// TIA Portal V20 export
FUNCTION "01 T4 LANT Alarms" : Void   // FC1112, LAD
TITLE = ALARMS
{ S7_Optimized_Access := 'TRUE' }
// stored: AutoNumber false, IsIECCheckEnabled true, SetENOAutomatically false
   VAR_TEMP
      Trash : Bool;
   END_VAR
BEGIN

REGION Network 1: ============ ALARMS RESET ============
END_REGION

REGION Network 2: Alarms Reset
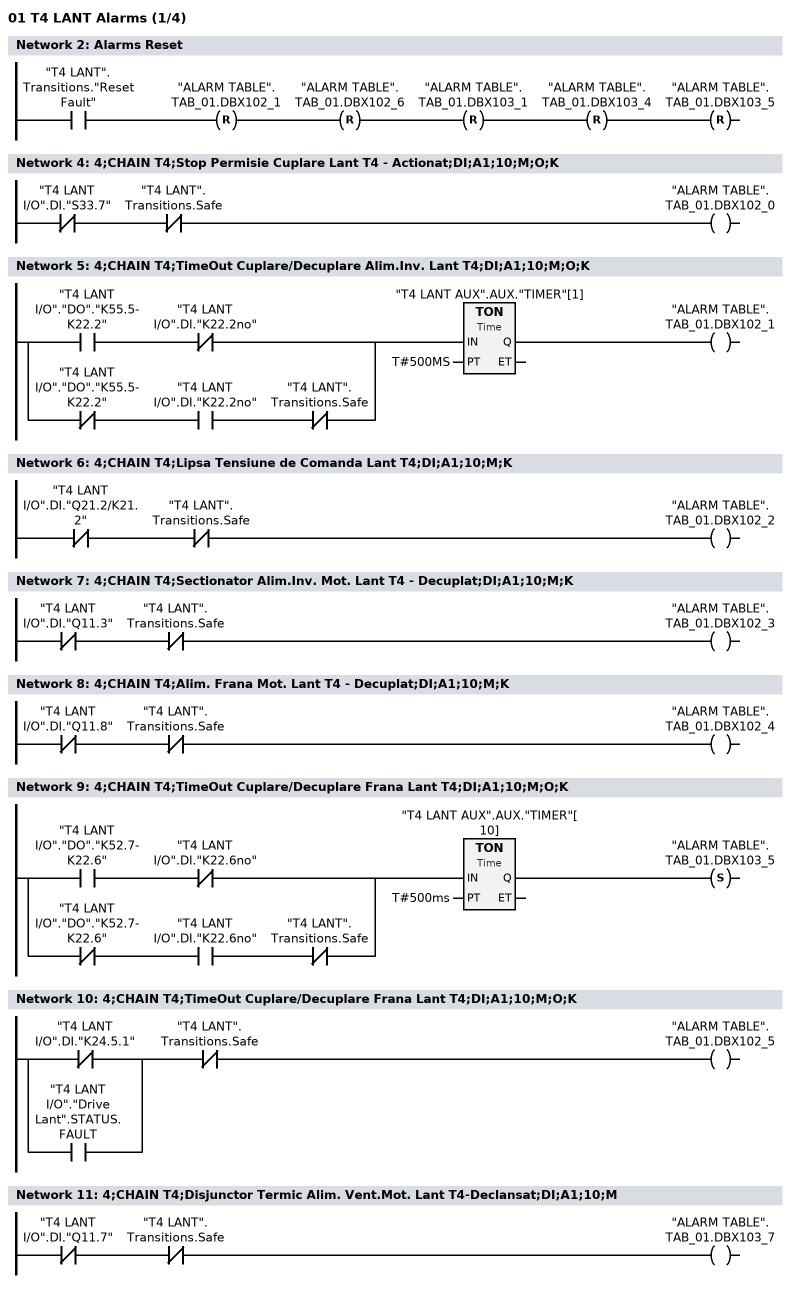
   RUNG wire#powerrail
      Contact( "T4 LANT".Transitions."Reset Fault" )
      R_Coil( "ALARM TABLE".TAB_01.DBX102_1 )
      R_Coil( "ALARM TABLE".TAB_01.DBX102_6 )
      R_Coil( "ALARM TABLE".TAB_01.DBX103_1 )
      R_Coil( "ALARM TABLE".TAB_01.DBX103_4 )
      R_Coil( "ALARM TABLE".TAB_01.DBX103_5 )
   END_RUNG
   // the same network as SCL:
   IF "T4 LANT".Transitions."Reset Fault" THEN
       "ALARM TABLE".TAB_01.DBX102_1 := FALSE;
       "ALARM TABLE".TAB_01.DBX102_6 := FALSE;
       "ALARM TABLE".TAB_01.DBX103_1 := FALSE;
       "ALARM TABLE".TAB_01.DBX103_4 := FALSE;
       "ALARM TABLE".TAB_01.DBX103_5 := FALSE;
   END_IF;
END_REGION

REGION Network 3: ============ PERMANENT CONDITIONS ============
END_REGION

REGION Network 4: 4;CHAIN T4;Stop Permisie Cuplare Lant T4 - Actionat;DI;A1;10;M;O;K
   RUNG wire#powerrail
      I_Contact( "T4 LANT I/O".DI."S33.7" )
      I_Contact( "T4 LANT".Transitions.Safe )
      Coil( "ALARM TABLE".TAB_01.DBX102_0 )
   END_RUNG
   // the same network as SCL:
   "ALARM TABLE".TAB_01.DBX102_0 := NOT "T4 LANT I/O".DI."S33.7" AND NOT "T4 LANT".Transitions.Safe;
END_REGION

REGION Network 5: 4;CHAIN T4;TimeOut Cuplare/Decuplare Alim.Inv. Lant T4;DI;A1;10;M;O;K
   RUNG wire#powerrail
      Contact( "T4 LANT I/O"."DO"."K55.5-K22.2" )
      I_Contact( "T4 LANT I/O".DI."K22.2no" )
      wire#w1
      { S7_Templates := "time_type := Time" } "T4 LANT AUX".AUX."TIMER"[1].TON(pt := T#500MS, et =>)
      Coil( "ALARM TABLE".TAB_01.DBX102_1 )
   END_RUNG
   RUNG wire#powerrail
      I_Contact( "T4 LANT I/O"."DO"."K55.5-K22.2" )
      Contact( "T4 LANT I/O".DI."K22.2no" )
      I_Contact( "T4 LANT".Transitions.Safe )
   END_RUNG wire#w1
   // the same network as SCL:
   "T4 LANT AUX".AUX."TIMER"[1].TON(IN := ("T4 LANT I/O"."DO"."K55.5-K22.2" AND NOT "T4 LANT I/O".DI."K22.2no") OR (NOT "T4 LANT I/O"."DO"."K55.5-K22.2" AND "T4 LANT I/O".DI."K22.2no" AND NOT "T4 LANT".Transitions.Safe),
                           PT := T#500MS);
   "ALARM TABLE".TAB_01.DBX102_1 := "T4 LANT AUX".AUX."TIMER"[1].Q;
END_REGION

REGION Network 6: 4;CHAIN T4;Lipsa Tensiune de Comanda Lant T4;DI;A1;10;M;K
   RUNG wire#powerrail
      I_Contact( "T4 LANT I/O".DI."Q21.2/K21.2" )
      I_Contact( "T4 LANT".Transitions.Safe )
      Coil( "ALARM TABLE".TAB_01.DBX102_2 )
   END_RUNG
   // the same network as SCL:
   "ALARM TABLE".TAB_01.DBX102_2 := NOT "T4 LANT I/O".DI."Q21.2/K21.2" AND NOT "T4 LANT".Transitions.Safe;
END_REGION

REGION Network 7: 4;CHAIN T4;Sectionator Alim.Inv. Mot. Lant T4 - Decuplat;DI;A1;10;M;K
   RUNG wire#powerrail
      I_Contact( "T4 LANT I/O".DI."Q11.3" )
      I_Contact( "T4 LANT".Transitions.Safe )
      Coil( "ALARM TABLE".TAB_01.DBX102_3 )
   END_RUNG
   // the same network as SCL:
   "ALARM TABLE".TAB_01.DBX102_3 := NOT "T4 LANT I/O".DI."Q11.3" AND NOT "T4 LANT".Transitions.Safe;
END_REGION

REGION Network 8: 4;CHAIN T4;Alim. Frana Mot. Lant T4 - Decuplat;DI;A1;10;M;K
   RUNG wire#powerrail
      I_Contact( "T4 LANT I/O".DI."Q11.8" )
      I_Contact( "T4 LANT".Transitions.Safe )
      Coil( "ALARM TABLE".TAB_01.DBX102_4 )
   END_RUNG
   // the same network as SCL:
   "ALARM TABLE".TAB_01.DBX102_4 := NOT "T4 LANT I/O".DI."Q11.8" AND NOT "T4 LANT".Transitions.Safe;
END_REGION

REGION Network 9: 4;CHAIN T4;TimeOut Cuplare/Decuplare Frana Lant T4;DI;A1;10;M;O;K
   RUNG wire#powerrail
      Contact( "T4 LANT I/O"."DO"."K52.7-K22.6" )
      I_Contact( "T4 LANT I/O".DI."K22.6no" )
      wire#w1
      { S7_Templates := "time_type := Time" } "T4 LANT AUX".AUX."TIMER"[10].TON(pt := T#500ms, et =>)
      S_Coil( "ALARM TABLE".TAB_01.DBX103_5 )
   END_RUNG
   RUNG wire#powerrail
      I_Contact( "T4 LANT I/O"."DO"."K52.7-K22.6" )
      Contact( "T4 LANT I/O".DI."K22.6no" )
      I_Contact( "T4 LANT".Transitions.Safe )
   END_RUNG wire#w1
   // the same network as SCL:
   "T4 LANT AUX".AUX."TIMER"[10].TON(IN := ("T4 LANT I/O"."DO"."K52.7-K22.6" AND NOT "T4 LANT I/O".DI."K22.6no") OR (NOT "T4 LANT I/O"."DO"."K52.7-K22.6" AND "T4 LANT I/O".DI."K22.6no" AND NOT "T4 LANT".Transitions.Safe),
                           PT := T#500ms);
   IF "T4 LANT AUX".AUX."TIMER"[10].Q THEN "ALARM TABLE".TAB_01.DBX103_5 := TRUE; END_IF;
END_REGION

REGION Network 10: 4;CHAIN T4;TimeOut Cuplare/Decuplare Frana Lant T4;DI;A1;10;M;O;K
   RUNG wire#powerrail
      I_Contact( "T4 LANT I/O".DI."K24.5.1" )
      wire#w1
      I_Contact( "T4 LANT".Transitions.Safe )
      Coil( "ALARM TABLE".TAB_01.DBX102_5 )
   END_RUNG
   RUNG wire#powerrail
      Contact( "T4 LANT I/O"."Drive Lant".STATUS.FAULT )
   END_RUNG wire#w1
   // the same network as SCL:
   "ALARM TABLE".TAB_01.DBX102_5 := (NOT "T4 LANT I/O".DI."K24.5.1" OR "T4 LANT I/O"."Drive Lant".STATUS.FAULT) AND NOT "T4 LANT".Transitions.Safe;
END_REGION

REGION Network 11: 4;CHAIN T4;Disjunctor Termic Alim. Vent.Mot. Lant T4-Declansat;DI;A1;10;M
   RUNG wire#powerrail
      I_Contact( "T4 LANT I/O".DI."Q11.7" )
      I_Contact( "T4 LANT".Transitions.Safe )
      Coil( "ALARM TABLE".TAB_01.DBX103_7 )
   END_RUNG
   // the same network as SCL:
   "ALARM TABLE".TAB_01.DBX103_7 := NOT "T4 LANT I/O".DI."Q11.7" AND NOT "T4 LANT".Transitions.Safe;
END_REGION

REGION Network 12: 4;CHAIN T4;Alim. Frana Mot. Lant T4 - Decuplat;DI;A1;10;M;K
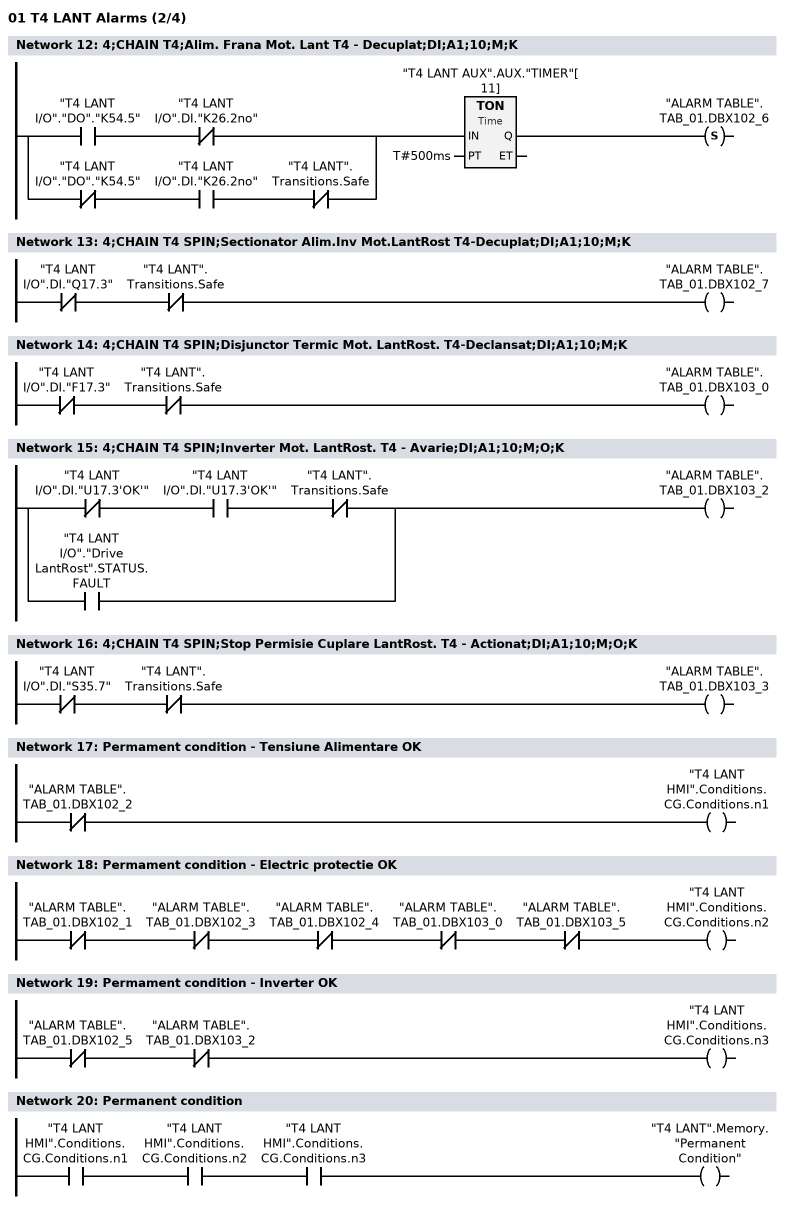
   RUNG wire#powerrail
      Contact( "T4 LANT I/O"."DO"."K54.5" )
      I_Contact( "T4 LANT I/O".DI."K26.2no" )
      wire#w1
      { S7_Templates := "time_type := Time" } "T4 LANT AUX".AUX."TIMER"[11].TON(pt := T#500ms, et =>)
      S_Coil( "ALARM TABLE".TAB_01.DBX102_6 )
   END_RUNG
   RUNG wire#powerrail
      I_Contact( "T4 LANT I/O"."DO"."K54.5" )
      Contact( "T4 LANT I/O".DI."K26.2no" )
      I_Contact( "T4 LANT".Transitions.Safe )
   END_RUNG wire#w1
   // the same network as SCL:
   "T4 LANT AUX".AUX."TIMER"[11].TON(IN := ("T4 LANT I/O"."DO"."K54.5" AND NOT "T4 LANT I/O".DI."K26.2no") OR (NOT "T4 LANT I/O"."DO"."K54.5" AND "T4 LANT I/O".DI."K26.2no" AND NOT "T4 LANT".Transitions.Safe),
                           PT := T#500ms);
   IF "T4 LANT AUX".AUX."TIMER"[11].Q THEN "ALARM TABLE".TAB_01.DBX102_6 := TRUE; END_IF;
END_REGION

REGION Network 13: 4;CHAIN T4 SPIN;Sectionator Alim.Inv Mot.LantRost T4-Decuplat;DI;A1;10;M;K
   RUNG wire#powerrail
      I_Contact( "T4 LANT I/O".DI."Q17.3" )
      I_Contact( "T4 LANT".Transitions.Safe )
      Coil( "ALARM TABLE".TAB_01.DBX102_7 )
   END_RUNG
   // the same network as SCL:
   "ALARM TABLE".TAB_01.DBX102_7 := NOT "T4 LANT I/O".DI."Q17.3" AND NOT "T4 LANT".Transitions.Safe;
END_REGION

REGION Network 14: 4;CHAIN T4 SPIN;Disjunctor Termic Mot. LantRost. T4-Declansat;DI;A1;10;M;K
   RUNG wire#powerrail
      I_Contact( "T4 LANT I/O".DI."F17.3" )
      I_Contact( "T4 LANT".Transitions.Safe )
      Coil( "ALARM TABLE".TAB_01.DBX103_0 )
   END_RUNG
   // the same network as SCL:
   "ALARM TABLE".TAB_01.DBX103_0 := NOT "T4 LANT I/O".DI."F17.3" AND NOT "T4 LANT".Transitions.Safe;
END_REGION

REGION Network 15: 4;CHAIN T4 SPIN;Inverter Mot. LantRost. T4 - Avarie;DI;A1;10;M;O;K
   RUNG wire#powerrail
      I_Contact( "T4 LANT I/O".DI."U17.3'OK'" )
      Contact( "T4 LANT I/O".DI."U17.3'OK'" )
      I_Contact( "T4 LANT".Transitions.Safe )
      wire#w1
      Coil( "ALARM TABLE".TAB_01.DBX103_2 )
   END_RUNG
   RUNG wire#powerrail
      Contact( "T4 LANT I/O"."Drive LantRost".STATUS.FAULT )
   END_RUNG wire#w1
   // the same network as SCL:
   "ALARM TABLE".TAB_01.DBX103_2 := (NOT "T4 LANT I/O".DI."U17.3'OK'" AND "T4 LANT I/O".DI."U17.3'OK'" AND NOT "T4 LANT".Transitions.Safe) OR "T4 LANT I/O"."Drive LantRost".STATUS.FAULT;
END_REGION

REGION Network 16: 4;CHAIN T4 SPIN;Stop Permisie Cuplare LantRost. T4 - Actionat;DI;A1;10;M;O;K
   RUNG wire#powerrail
      I_Contact( "T4 LANT I/O".DI."S35.7" )
      I_Contact( "T4 LANT".Transitions.Safe )
      Coil( "ALARM TABLE".TAB_01.DBX103_3 )
   END_RUNG
   // the same network as SCL:
   "ALARM TABLE".TAB_01.DBX103_3 := NOT "T4 LANT I/O".DI."S35.7" AND NOT "T4 LANT".Transitions.Safe;
END_REGION

REGION Network 17: Permament condition - Tensiune Alimentare OK
   RUNG wire#powerrail
      I_Contact( "ALARM TABLE".TAB_01.DBX102_2 )
      Coil( "T4 LANT HMI".Conditions.CG.Conditions.n1 )
   END_RUNG
   // the same network as SCL:
   "T4 LANT HMI".Conditions.CG.Conditions.n1 := NOT "ALARM TABLE".TAB_01.DBX102_2;
END_REGION

REGION Network 18: Permament condition - Electric protectie OK
   RUNG wire#powerrail
      I_Contact( "ALARM TABLE".TAB_01.DBX102_1 )
      I_Contact( "ALARM TABLE".TAB_01.DBX102_3 )
      I_Contact( "ALARM TABLE".TAB_01.DBX102_4 )
      I_Contact( "ALARM TABLE".TAB_01.DBX103_0 )
      I_Contact( "ALARM TABLE".TAB_01.DBX103_5 )
      Coil( "T4 LANT HMI".Conditions.CG.Conditions.n2 )
   END_RUNG
   // the same network as SCL:
   "T4 LANT HMI".Conditions.CG.Conditions.n2 := NOT "ALARM TABLE".TAB_01.DBX102_1 AND NOT "ALARM TABLE".TAB_01.DBX102_3 AND NOT "ALARM TABLE".TAB_01.DBX102_4 AND NOT "ALARM TABLE".TAB_01.DBX103_0 AND NOT "ALARM TABLE".TAB_01.DBX103_5;
END_REGION

REGION Network 19: Permament condition - Inverter OK
   RUNG wire#powerrail
      I_Contact( "ALARM TABLE".TAB_01.DBX102_5 )
      I_Contact( "ALARM TABLE".TAB_01.DBX103_2 )
      Coil( "T4 LANT HMI".Conditions.CG.Conditions.n3 )
   END_RUNG
   // the same network as SCL:
   "T4 LANT HMI".Conditions.CG.Conditions.n3 := NOT "ALARM TABLE".TAB_01.DBX102_5 AND NOT "ALARM TABLE".TAB_01.DBX103_2;
END_REGION

REGION Network 20: Permanent condition
   RUNG wire#powerrail
      Contact( "T4 LANT HMI".Conditions.CG.Conditions.n1 )
      Contact( "T4 LANT HMI".Conditions.CG.Conditions.n2 )
      Contact( "T4 LANT HMI".Conditions.CG.Conditions.n3 )
      Coil( "T4 LANT".Memory."Permanent Condition" )
   END_RUNG
   // the same network as SCL:
   "T4 LANT".Memory."Permanent Condition" := "T4 LANT HMI".Conditions.CG.Conditions.n1 AND "T4 LANT HMI".Conditions.CG.Conditions.n2 AND "T4 LANT HMI".Conditions.CG.Conditions.n3;
END_REGION

REGION Network 21: ======= MACHINE MOVEMENT CONTROL (SENSORS / ENCODERS / INTERLOCKS) =======
END_REGION

REGION Network 22: 4;CHAIN T4;TimeOut Deplasare Lant T4 in pozitia Pas;DI;A1;10;M;O;K
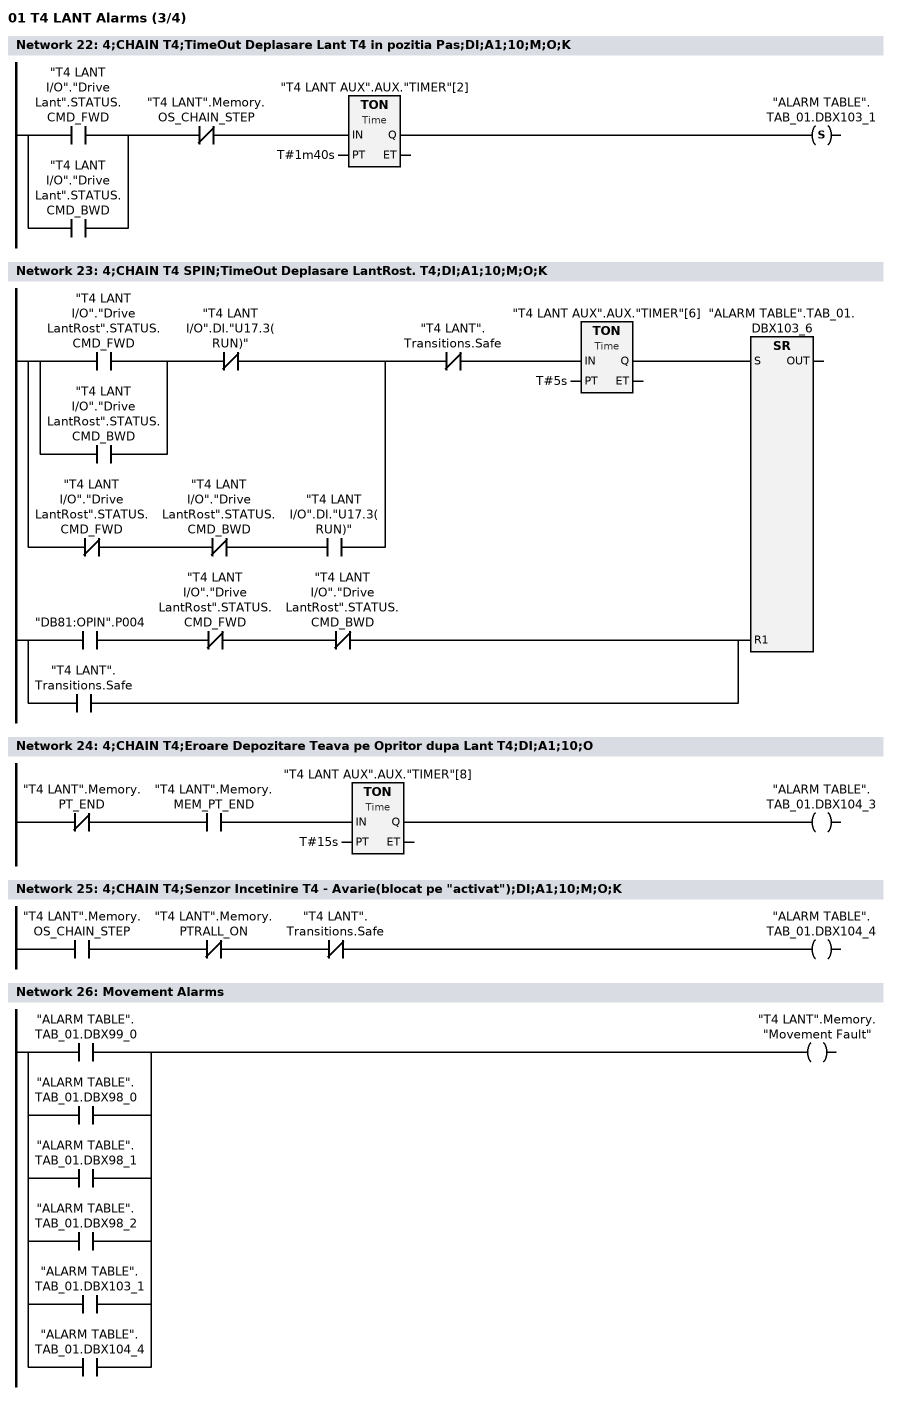
   RUNG wire#powerrail
      Contact( "T4 LANT I/O"."Drive Lant".STATUS.CMD_FWD )
      wire#w1
      I_Contact( "T4 LANT".Memory.OS_CHAIN_STEP )
      { S7_Templates := "time_type := Time" } "T4 LANT AUX".AUX."TIMER"[2].TON(pt := T#1m40s, et =>)
      S_Coil( "ALARM TABLE".TAB_01.DBX103_1 )
   END_RUNG
   RUNG wire#powerrail
      Contact( "T4 LANT I/O"."Drive Lant".STATUS.CMD_BWD )
   END_RUNG wire#w1
   // the same network as SCL:
   "T4 LANT AUX".AUX."TIMER"[2].TON(IN := ("T4 LANT I/O"."Drive Lant".STATUS.CMD_FWD OR "T4 LANT I/O"."Drive Lant".STATUS.CMD_BWD) AND NOT "T4 LANT".Memory.OS_CHAIN_STEP,
                           PT := T#1m40s);
   IF "T4 LANT AUX".AUX."TIMER"[2].Q THEN "ALARM TABLE".TAB_01.DBX103_1 := TRUE; END_IF;
END_REGION

REGION Network 23: 4;CHAIN T4 SPIN;TimeOut Deplasare LantRost. T4;DI;A1;10;M;O;K
   RUNG wire#powerrail
      Contact( "T4 LANT I/O"."Drive LantRost".STATUS.CMD_FWD )
      wire#w1
      I_Contact( "T4 LANT I/O".DI."U17.3(RUN)" )
      wire#w2
      I_Contact( "T4 LANT".Transitions.Safe )
      { S7_Templates := "time_type := Time" } "T4 LANT AUX".AUX."TIMER"[6].TON(pt := T#5s, et =>)
      S_SR(operand := "ALARM TABLE".TAB_01.DBX103_6, r1 := wire#w3)
   END_RUNG
   RUNG wire#powerrail
      Contact( "T4 LANT I/O"."Drive LantRost".STATUS.CMD_BWD )
   END_RUNG wire#w1
   RUNG wire#powerrail
      I_Contact( "T4 LANT I/O"."Drive LantRost".STATUS.CMD_FWD )
      I_Contact( "T4 LANT I/O"."Drive LantRost".STATUS.CMD_BWD )
      Contact( "T4 LANT I/O".DI."U17.3(RUN)" )
   END_RUNG wire#w2
   RUNG wire#powerrail
      Contact( "DB81:OPIN".P004 )
      I_Contact( "T4 LANT I/O"."Drive LantRost".STATUS.CMD_FWD )
      I_Contact( "T4 LANT I/O"."Drive LantRost".STATUS.CMD_BWD )
   END_RUNG wire#w3
   RUNG wire#powerrail
      Contact( "T4 LANT".Transitions.Safe )
   END_RUNG wire#w3
   // the same network as SCL:
   "T4 LANT AUX".AUX."TIMER"[6].TON(IN := ((("T4 LANT I/O"."Drive LantRost".STATUS.CMD_FWD OR "T4 LANT I/O"."Drive LantRost".STATUS.CMD_BWD) AND NOT "T4 LANT I/O".DI."U17.3(RUN)") OR (NOT "T4 LANT I/O"."Drive LantRost".STATUS.CMD_FWD AND NOT "T4 LANT I/O"."Drive LantRost".STATUS.CMD_BWD AND "T4 LANT I/O".DI."U17.3(RUN)")) AND NOT "T4 LANT".Transitions.Safe,
                           PT := T#5s);
   IF "T4 LANT AUX".AUX."TIMER"[6].Q THEN
       "ALARM TABLE".TAB_01.DBX103_6 := TRUE;   // SR flip-flop
   END_IF;
   IF ("DB81:OPIN".P004 AND NOT "T4 LANT I/O"."Drive LantRost".STATUS.CMD_FWD AND NOT "T4 LANT I/O"."Drive LantRost".STATUS.CMD_BWD) OR "T4 LANT".Transitions.Safe THEN
       "ALARM TABLE".TAB_01.DBX103_6 := FALSE;
   END_IF;
END_REGION

REGION Network 24: 4;CHAIN T4;Eroare Depozitare Teava pe Opritor dupa Lant T4;DI;A1;10;O
   RUNG wire#powerrail
      I_Contact( "T4 LANT".Memory.PT_END )
      Contact( "T4 LANT".Memory.MEM_PT_END )
      { S7_Templates := "time_type := Time" } "T4 LANT AUX".AUX."TIMER"[8].TON(pt := T#15s, et =>)
      Coil( "ALARM TABLE".TAB_01.DBX104_3 )
   END_RUNG
   // the same network as SCL:
   "T4 LANT AUX".AUX."TIMER"[8].TON(IN := NOT "T4 LANT".Memory.PT_END AND "T4 LANT".Memory.MEM_PT_END,
                           PT := T#15s);
   "ALARM TABLE".TAB_01.DBX104_3 := "T4 LANT AUX".AUX."TIMER"[8].Q;
END_REGION

REGION Network 25: 4;CHAIN T4;Senzor Incetinire T4 - Avarie(blocat pe "activat");DI;A1;10;M;O;K
   RUNG wire#powerrail
      Contact( "T4 LANT".Memory.OS_CHAIN_STEP )
      I_Contact( "T4 LANT".Memory.PTRALL_ON )
      I_Contact( "T4 LANT".Transitions.Safe )
      Coil( "ALARM TABLE".TAB_01.DBX104_4 )
   END_RUNG
   // the same network as SCL:
   "ALARM TABLE".TAB_01.DBX104_4 := "T4 LANT".Memory.OS_CHAIN_STEP AND NOT "T4 LANT".Memory.PTRALL_ON AND NOT "T4 LANT".Transitions.Safe;
END_REGION

REGION Network 26: Movement Alarms
   RUNG wire#powerrail
      Contact( "ALARM TABLE".TAB_01.DBX99_0 )
      wire#w1
      Coil( "T4 LANT".Memory."Movement Fault" )
   END_RUNG
   RUNG wire#powerrail
      Contact( "ALARM TABLE".TAB_01.DBX98_0 )
   END_RUNG wire#w1
   RUNG wire#powerrail
      Contact( "ALARM TABLE".TAB_01.DBX98_1 )
   END_RUNG wire#w1
   RUNG wire#powerrail
      Contact( "ALARM TABLE".TAB_01.DBX98_2 )
   END_RUNG wire#w1
   RUNG wire#powerrail
      Contact( "ALARM TABLE".TAB_01.DBX103_1 )
   END_RUNG wire#w1
   RUNG wire#powerrail
      Contact( "ALARM TABLE".TAB_01.DBX104_4 )
   END_RUNG wire#w1
   // the same network as SCL:
   "T4 LANT".Memory."Movement Fault" := "ALARM TABLE".TAB_01.DBX99_0 OR "ALARM TABLE".TAB_01.DBX98_0 OR "ALARM TABLE".TAB_01.DBX98_1 OR "ALARM TABLE".TAB_01.DBX98_2 OR "ALARM TABLE".TAB_01.DBX103_1 OR "ALARM TABLE".TAB_01.DBX104_4;
END_REGION

REGION Network 27: ======= OTHER ALARMS =======
END_REGION

REGION Network 28: ======= FAULT =======
END_REGION

REGION Network 29: Fault Transition
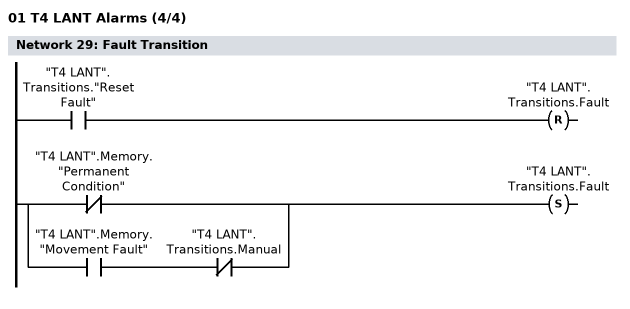
   RUNG wire#powerrail
      Contact( "T4 LANT".Transitions."Reset Fault" )
      R_Coil( "T4 LANT".Transitions.Fault )
   END_RUNG
   RUNG wire#powerrail
      I_Contact( "T4 LANT".Memory."Permanent Condition" )
      wire#w1
      S_Coil( "T4 LANT".Transitions.Fault )
   END_RUNG
   RUNG wire#powerrail
      Contact( "T4 LANT".Memory."Movement Fault" )
      I_Contact( "T4 LANT".Transitions.Manual )
   END_RUNG wire#w1
   // the same network as SCL:
   IF "T4 LANT".Transitions."Reset Fault" THEN "T4 LANT".Transitions.Fault := FALSE; END_IF;
   IF NOT "T4 LANT".Memory."Permanent Condition" OR ("T4 LANT".Memory."Movement Fault" AND NOT "T4 LANT".Transitions.Manual) THEN
       "T4 LANT".Transitions.Fault := TRUE;
   END_IF;
END_REGION
END_FUNCTION
